FUNCTION_BLOCK FloorSensors (* Composite Function Block Type *)
  (* Standard: 61499-2 *)
  (* Version 0.0, 7/12/2016, Andrei, nxtControl GmbH, template *)
  PACKAGE Main;
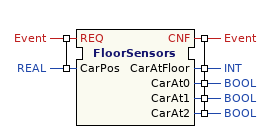
  EVENT_INPUT
    REQ WITH CarPos; (* Normal Execution Request *)
  END_EVENT
  EVENT_OUTPUT
    CNF WITH CarAtFloor, CarAt0, CarAt1, CarAt2; (* Execution Confirmation *)
  END_EVENT
  VAR_INPUT
    CarPos : REAL; (* Input event qualifier *)
  END_VAR
  VAR_OUTPUT
    CarAtFloor : INT; (* Output event qualifier *)
    CarAt0 : BOOL;
    CarAt1 : BOOL;
    CarAt2 : BOOL;
  END_VAR
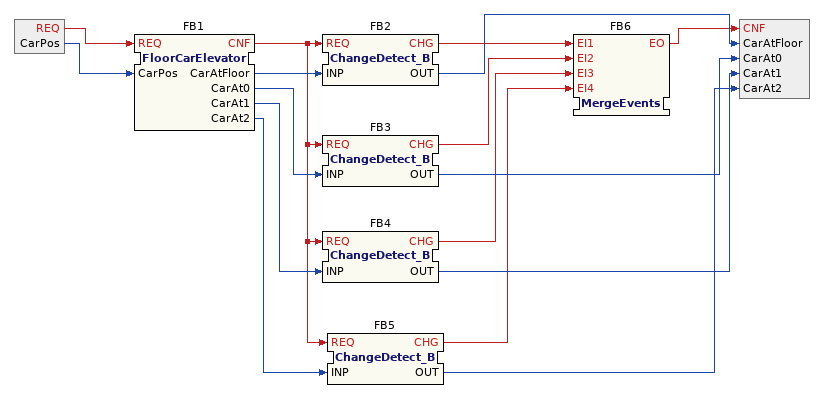
  FBS
    FB1 : FloorCarElevator;
    FB2 : ChangeDetect_B;
    FB3 : ChangeDetect_B;
    FB4 : ChangeDetect_B;
    FB5 : ChangeDetect_B;
    FB6 : MergeEvents;
  END_FBS
  EVENT_CONNECTIONS
    FB1.CNF TO FB2.REQ;
    FB1.CNF TO FB3.REQ;
    FB1.CNF TO FB4.REQ;
    FB1.CNF TO FB5.REQ;
    FB2.CHG TO FB6.EI1;
    FB3.CHG TO FB6.EI2;
    FB4.CHG TO FB6.EI3;
    FB5.CHG TO FB6.EI4;
    REQ TO FB1.REQ;
    FB6.EO TO CNF;
  END_CONNECTIONS
  DATA_CONNECTIONS
    FB1.CarAtFloor TO FB2.INP;
    FB1.CarAt0 TO FB3.INP;
    FB1.CarAt1 TO FB4.INP;
    FB1.CarAt2 TO FB5.INP;
    FB4.OUT TO CarAt1;
    FB5.OUT TO CarAt2;
    FB3.OUT TO CarAt0;
    FB2.OUT TO CarAtFloor;
    CarPos TO FB1.CarPos;
  END_CONNECTIONS
END_FUNCTION_BLOCK
